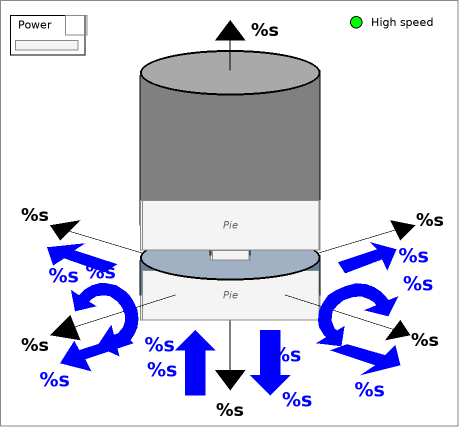
VISUALIZATION VISU_M2Figure  // 459x427
VAR_IN_OUT
	ref : M2;
    widget : M2FigureWidget;
END_VAR
    RoundedRectangle (10,15 75x40)
    Line (395,230) (295,260)
    Line (165,260) (65,230)
    Line (230,370) (230,300)
    Pie (140,270 180x50)
    Rectangle (140,260 180x35)
    Pie (142,270 177x50)
    Ellipse (140,235 180x45)
    Line (320,295) (320,255)
    Line (140,295) (140,260)
    Rectangle (140,75 180x150)
    Ellipse (140,50 180x45)
    Line (320,225) (320,70)
    Line (140,225) (140,75)
    Pie (210,250 40x10)
    Rectangle (210,235 40x20)
    Pie (212,250 37x10)
    Line (250,255) (250,235)
    Line (210,255) (210,235)
    Pie (140,200 180x50)
    Pie (142,200 177x50)
    Line (230,70) (230,35)
    Polygon (215,40) (230,20) (245,40), invisible if: widget.a_top_head_invisible
    Line (395,330) (285,295)
    Line (175,295) (65,330)
    Polygon (410,335) (400,320) (385,340), invisible if: widget.c_right_head_invisible
    Polygon (415,225) (390,220) (400,240), invisible if: widget.c_right_head_invisible
    Rectangle (250,15 30x30), "%s", tooltip "The Z axis", text variable: widget.a_top_name, invisible if: widget.a_top_head_invisible
    Rectangle (410,325 30x30), "%s", tooltip "The Z axis", text variable: widget.c_right_name, invisible if: widget.c_right_head_invisible
    Rectangle (415,205 30x30), "%s", tooltip "The Z axis", text variable: widget.b_right_name, invisible if: widget.c_right_head_invisible
    Polygon (330,350) (347,344) (385,355) (395,345) (400,365) (360,375) (375,365), invisible if: widget.c_right_arrow_invisible
    Polygon (104,272) (117,264) (74,250) (85,243) (47,247) (53,265) (64,258), invisible if: widget.c_left_arrow_invisible
    Polygon (110,336) (115,347) (123,345) (130,340) (134,334) (137,327) (138,319) (137,310) (133,301) (129,295) (125,291) (116,285) (106,283) (99,283) (92,285) (85,289) (78,296) (86,304) (91,299) (96,296) (104,295) (110,296) (117,301) (122,307) (125,315) (125,321) (123,327) (118,333), invisible if: widget.e_arrow_invisible
    Rectangle (350,375 40x30), "%s", tooltip "The Z axis", text variable: widget.c_right_arrow_name, invisible if: widget.c_right_arrow_invisible
    Rectangle (44,261 40x30), "%s", tooltip "The Z axis", text variable: widget.c_left_arrow_name, invisible if: widget.c_left_arrow_invisible
    Polygon (75,311) (71,290) (96,306), invisible if: widget.e_left_arrow_invisible
    Polygon (97,346) (111,325) (119,356), invisible if: widget.e_right_arrow_invisible
    Polygon (379,312) (390,308) (389,301) (385,296) (380,291) (374,287) (366,284) (356,283) (345,286) (336,290) (328,295) (322,304) (319,311) (318,320) (319,327) (324,335) (330,340) (340,333) (334,328) (331,320) (332,311) (337,305) (343,300) (352,297) (361,296) (369,299) (374,302) (377,306), invisible if: widget.d_arrow_invisible
    Polygon (364,310) (398,296) (388,316), invisible if: widget.d_right_arrow_invisible
    Polygon (316,343) (344,326) (341,346), invisible if: widget.d_left_arrow_invisible
    Rectangle (380,269 77x30), "%s", tooltip "The Z axis", text variable: widget.d_right_arrow_name, invisible if: widget.d_right_arrow_invisible
    Rectangle (248,340 77x30), "%s", tooltip "The Z axis", text variable: widget.d_left_arrow_name, invisible if: widget.d_left_arrow_invisible
    Polygon (345,273) (338,262) (377,249) (370,242) (396,249) (387,270) (382,259), invisible if: widget.b_right_arrow_invisible
    Rectangle (394,241 40x30), "%s", tooltip "The Z axis", text variable: widget.b_right_arrow_name, invisible if: widget.b_right_arrow_invisible
    Polygon (133,343) (125,335) (79,350) (74,341) (60,363) (91,371) (85,359), invisible if: widget.b_left_arrow_invisible
    Rectangle (35,365 40x30), "%s", tooltip "The Z axis", text variable: widget.b_left_arrow_name, invisible if: widget.b_left_arrow_invisible
    Rectangle (65,257 72x30), "%s", tooltip "The Z axis", text variable: widget.e_left_arrow_name, invisible if: widget.e_left_arrow_invisible
    Rectangle (124,330 72x30), "%s", tooltip "The Z axis", text variable: widget.e_right_arrow_name, invisible if: widget.e_right_arrow_invisible
    Polygon (205,395) (185,395) (185,350) (175,350) (195,330) (215,350) (205,350), invisible if: widget.a_top_arrow_invisible
    Rectangle (140,355 45x30), "%s", tooltip "The Z axis", text variable: widget.a_top_arrow_name, invisible if: widget.a_top_arrow_invisible
    Polygon (280,330) (260,330) (260,375) (250,375) (270,395) (290,375) (280,375), invisible if: widget.a_bottom_arrow_invisible
    Polygon (215,370) (230,390) (245,370), invisible if: widget.a_bottom_head_invisible
    Rectangle (275,385 45x30), "%s", tooltip "The Z axis", text variable: widget.a_bottom_arrow_name, invisible if: widget.a_bottom_arrow_invisible
    Rectangle (215,395 30x30), "%s", tooltip "The Z axis", text variable: widget.a_bottom_name, invisible if: widget.a_bottom_head_invisible
    Polygon (50,225) (80,220) (60,240), invisible if: widget.c_left_head_invisible
    Polygon (50,335) (70,315) (80,340), invisible if: widget.b_left_head_invisible
    Rectangle (20,330 30x30), "%s", tooltip "The Z axis", text variable: widget.b_left_name, invisible if: widget.b_left_head_invisible
    Rectangle (20,200 30x30), "%s", tooltip "The Z axis", text variable: widget.c_left_name, invisible if: widget.c_left_head_invisible
    Progressbar (15,40 63x10), variable: widget.power_percent
    Label (15,10 50x30), "Power"
    Frame (65,15 22x20)
        shows VISU_State_gray_green(state := widget.power_on)
    Ellipse (350,16 12x12), invisible if: widget.high_speed_invisible
    Label (368,10 70x25), "High speed", invisible if: widget.high_speed_invisible
END_VISUALIZATION

(* stored: Version 1.1.0.1, ProductVersion 3.1.4019.2
   Visu VISU_M2Figure: Id {c09ec73c-2660-413a-a8df-2e24aceb8f37} *)
